// TIA Portal V17 export
// export: Created 2024-09-15T12:30:32.0507044Z, ExportSetting WithDefaults, DisplayName Totally Integrated Automation Portal, DisplayVersion V17, DisplayName TIA Portal Openness, DisplayVersion V17, DisplayName TIA Portal Version Control Interface, DisplayVersion V17, DisplayName STEP 7 Professional, DisplayVersion V17, DisplayName STEP 7 Safety, DisplayVersion V17, DisplayName WinCC Professional, DisplayVersion V17
TYPE "typ_Camera_Picture"
// stored: IsFailsafeCompliant false
   STRUCT
      ldt_ts : LDT;
      s_data : String;
   END_STRUCT;
END_TYPE
